FUNCTION_BLOCK FB_RampGeneration
VAR_INPUT
RampStart : REAL ; //Start value of ramp
RampTarget : REAL ; //Target Value of ramp
RampTimeStep : REAL ; //100ms call
RampFactor : REAL ; //Units added
END_VAR

VAR_OUTPUT
RampOutput : REAL ;
END_VAR

IF RampStart < RampTarget THEN
	RampStart := RampStart + (RampFactor * RampTimeStep) ;
	IF (RampStart > RampTarget) THEN
		RampStart := RampTarget ;
	END_IF
END_IF 

IF RampStart > RampTarget THEN  
	RampStart := RampStart - (RampFactor * RampTimeStep) ;
	IF (RampStart < RampTarget) THEN
		RampStart := RampTarget;
	END_IF
END_IF

RampOutput := RampStart ;

END_FUNCTION_BLOCK

(* stored: Version 1.1.0.1, ProductVersion 3.1.4024.12
   POU FB_RampGeneration: Id {b326c7de-8336-4158-9951-98f1784e2af3}, SpecialFunc None *)
